// TIA Portal V19 export
TYPE "OOAx_Sts"
// stored: Access Published
   STRUCT
      AlarmPresence : Bool;   // Cumulative alarm presence
      WarningPresence : Bool;   // Cumulative warning presence
      StandStill : Bool;   // Axis is standstill
      Homed : Bool;   // Axis is homed
      HomingPermitted : Bool;
      HomingDone : Bool;
      MoveMinusPermitted : Bool;
      MovePlusPermitted : Bool;
      MoveAbsPermitted : Bool;
      Positioned : Bool;   // On when move abs command is on and axis is in position
      InPosition : Bool;   // Always on when axis in in target position
      IsAtMinusLimit : Bool;   // Axis is at SW or HWD limit minus
      IsAtPlusLimit : Bool;   // Axis is at SW or HWD limit plus
      ActualPosition : LReal;   // mm
      ActualSpeed : LReal;   // xxxx : Depend from VelocityMeasUnit
   END_STRUCT;
END_TYPE
